FUNCTION_BLOCK Heating_Ctx_Hmi
VAR_INPUT
	sStatusText				: Str;
	nStatusColor			: LWORD;
	
	bButton					: BOOL;
	sButtonText				: Str;
	nButtonColor			: LWORD;	
END_VAR

END_FUNCTION_BLOCK

(* stored: Version 1.1.0.1
   POU Heating_Ctx_Hmi: Id {73b31336-e86f-44f2-a942-2796c435ebeb}, SpecialFunc None *)
